// TIA Portal V19 export
DATA_BLOCK "Top_Valve_Control"   // DB3
// stored: InstanceOfName Vavle_Control, InstanceOfType FB
"Vavle_Control"
   // VAR_INPUT
   //    Closed : Bool;
   //    Open : Bool;
   //    OpenValve : Bool;
   // END_VAR
   // VAR_OUTPUT
   //    Actuator : Bool;
   //    State : String;
   // END_VAR
BEGIN
END_DATA_BLOCK
